{attribute 'qualified_only'}
{attribute 'strict'}
TYPE E_MachineState :
(
	SYSTEM_POWER_UP			,
	STOPPED					,
	SYSTEM_INITIALISING		,
	SYSTEM_READY_TO_START	,
	SYSTEM_AUTO_CYCLE		,
	STOPPING				,
	MANUAL_MODE				,
	FAULT					,
	SAFETY
);
END_TYPE

(* stored: Version 1.1.0.1, ProductVersion 3.1.4026.17
   DUT E_MachineState: Id {36ef2dd6-2a0f-4be1-8e2a-d44a3a1a5753} *)
